FUNCTION_BLOCK EnableSequence_TestSuite
VAR
	ThisTestSuite : TestSuite<TestSuiteParameter.MaxTestCount>('C:\ProgramData\Beckhoff\TwinCAT\3.1\Boot\EnableSequence_Tests.xml') := (TestSuiteName := 'EnableSequence Test Suite');
END_VAR

SequenceAcceptsEnableCommand_Test();
SequenceRejectsCommandWithNoAxes_Test();
SequenceRejectsCommandWithNoCAGroup_Test();
SequenceRejectsDuplicateCommand_Test();
SequenceAcceptsMover_Test();
SequenceRejectsNullMoverRegister_Test();
SequenceReportsCorrectMoverNumber_Test();

METHOD SequenceAcceptsEnableCommand_Test : BOOL
VAR
	stubCAGroup : CollisionGroup;
	stubMover : XtsMover;
	EnableSequence : XtsEnableSequence := (MyCollisionGroup := stubCAGroup);
	Expected : BOOL := TRUE;
	Actual	 : BOOL;
END_VAR
IF ThisTestSuite.Test(__POUNAME()).ExecuteTest() THEN
	EnableSequence.RegisterMovers(stubMover);
	Actual := SUCCEEDED(EnableSequence.Enable());
	ThisTestSuite.Test(__POUNAME()).AssertEqual(Expected, Actual);
END_IF
END_METHOD

METHOD SequenceAcceptsMover_Test : BOOL
VAR
	stubCAGroup : CollisionGroup;
	stub_Mover : XtsMover;
	EnableSequence : XtsEnableSequence := (MyCollisionGroup := stubCAGroup);
	Expected : BOOL := TRUE;
	Actual	 : BOOL;
END_VAR
IF ThisTestSuite.Test(__POUNAME()).ExecuteTest() THEN
	EnableSequence.RegisterMovers(stub_Mover);
	Actual := SUCCEEDED(EnableSequence.Enable());
	ThisTestSuite.Test(__POUNAME()).AssertEqual(Expected, Actual);
END_IF
END_METHOD

METHOD SequenceRejectsCommandWithNoAxes_Test : BOOL
VAR
		stubCAGroup : CollisionGroup;
	EnableSequence : XtsEnableSequence := (MyCollisionGroup := stubCAGroup);
	Expected : BOOL := TRUE;
	Actual	 : BOOL;
END_VAR
IF ThisTestSuite.Test(__POUNAME()).ExecuteTest() THEN
	Actual := FAILED(EnableSequence.Enable());
	ThisTestSuite.Test(__POUNAME()).AssertEqual(Expected, Actual);
END_IF
END_METHOD

METHOD SequenceRejectsCommandWithNoCAGroup_Test : BOOL
VAR
	EnableSequence : XtsEnableSequence;
	Expected : BOOL := TRUE;
	Actual	 : BOOL;
END_VAR
IF ThisTestSuite.Test(__POUNAME()).ExecuteTest() THEN
	Actual := FAILED(EnableSequence.Enable());
	ThisTestSuite.Test(__POUNAME()).AssertEqual(Expected, Actual);
END_IF
END_METHOD

METHOD SequenceRejectsDuplicateCommand_Test : BOOL
VAR
	stubCAGroup : CollisionGroup;
	EnableSequence : XtsEnableSequence := (MyCollisionGroup := stubCAGroup);
	Expected : BOOL := TRUE;
	Actual	 : BOOL;
END_VAR
IF ThisTestSuite.Test(__POUNAME()).ExecuteTest() THEN
	EnableSequence.Enable();
	Actual := FAILED(EnableSequence.Enable());
	ThisTestSuite.Test(__POUNAME()).AssertEqual(Expected, Actual);
END_IF
END_METHOD

METHOD SequenceRejectsNullMoverRegister_Test
VAR
	stub_Mover : I_XtsMover;
	EnableSequence : XtsEnableSequence;
	Expected : BOOL := TRUE;
	Actual	 : BOOL;
END_VAR
IF ThisTestSuite.Test(__POUNAME()).ExecuteTest() THEN
	Actual := FAILED(EnableSequence.RegisterMovers(stub_Mover));
	ThisTestSuite.Test(__POUNAME()).AssertEqual(Expected, Actual);
END_IF
END_METHOD

METHOD SequenceReportsCorrectMoverNumber_Test : BOOL
VAR
	stubCAGroup : CollisionGroup;
	stub_Mover1 : stubMover;
	stub_Mover2 : stubMover;
	stub_Mover3 : stubMover;
	EnableSequence : XtsEnableSequence := (MyCollisionGroup := stubCAGroup);
	Expected : BOOL := TRUE;
	Actual	 : BOOL;
END_VAR
IF ThisTestSuite.Test(__POUNAME()).ExecuteTest() THEN
	EnableSequence.RegisterMovers(stub_Mover1);
	EnableSequence.RegisterMovers(stub_Mover2);
	EnableSequence.RegisterMovers(stub_Mover3);
	Actual := EnableSequence.RegisteredMoverNumber = 3;
	ThisTestSuite.Test(__POUNAME()).AssertEqual(Expected, Actual);
END_IF
END_METHOD

END_FUNCTION_BLOCK

(* stored: Version 1.1.0.1
   POU EnableSequence_TestSuite: Id {0a7c423d-1ec1-40a1-84cd-1f7627cf2709}, SpecialFunc None
   Method SequenceAcceptsEnableCommand_Test: Id {d8f7a973-bbd5-4c8b-b462-c79ceb666984}
   Method SequenceAcceptsMover_Test: Id {e91a3164-80ca-4533-820c-a6b0c8f9e00c}
   Method SequenceRejectsCommandWithNoAxes_Test: Id {9fde4aaf-da0d-421e-9b7a-9666ee182b4f}
   Method SequenceRejectsCommandWithNoCAGroup_Test: Id {bb0bce4d-8922-4996-9551-55aafd4891a1}
   Method SequenceRejectsDuplicateCommand_Test: Id {dfff0d2b-4c84-4d2f-bcd5-ddbfacfc030e}
   Method SequenceRejectsNullMoverRegister_Test: Id {8a9fa3df-ea12-4bf8-957f-b81e6275d244}
   Method SequenceReportsCorrectMoverNumber_Test: Id {98aae470-b0db-41b9-8128-0a32e5302399} *)
